// TwinCAT 3 PLC project Untitled1
// ProgramVersion: 3.1.4024.0
// libraries:
//   SysProcess, * (System)
//   Tc2_MC2, * (Beckhoff Automation GmbH)
//   Tc2_Standard, * (Beckhoff Automation GmbH)
//   Tc2_System, * (Beckhoff Automation GmbH)
//   Tc3_MC2_AdvancedHoming, * (Beckhoff Automation GmbH)
//   Tc3_Module, * (Beckhoff Automation GmbH)
//   VisuSymbols,3.5.10.0,System
// project tree:
//   DUTs/ ST_OPCUA.TcDUT
//   / GlobalTextList.TcGTLO, PlcTask.TcTTO, Visualization Manager.TcVMO (not stored)
//   GVLs/ GVL.TcGVL, IO.TcGVL
//   POUs/ Axis.TcPOU, MAIN.TcPOU, POU.TcPOU, process.TcPOU
//   VISUs/ Visualization.TcVIS
// real-time tasks:
//   TASK PlcTask: cycle T#10ms, priority 20, ADS port 350
// motion (NC):
//   TASK NC-Task 1 SAF: cycle T#2ms, priority 4, ADS port 501
//   TASK NC-Task 1 SVB: cycle T#10ms, priority 8, ADS port 511
//   AXIS Axis 1 (id 1)
//     OtherSettings: AllowMotionCmdToSlave=true
//     encoder EncType=1
//     drive DrvType=5
//       Analog: TorqueSetpointScale=10, ScaleFactorActTorque=0.1
//       TimeComp: TaskDelayCycles=1
//     controller CtrType=1
//       CtrPara: PriorControlFactor=1
//         Observer: BandWidth=20
//   AXIS linear Axis 3 (id 3)
//     Dynamic: AccelerationMaximum=50, DecelerationMaximum=50, Acceleration=25, Deceleration=25, Jerk=1211.25
//     Velo: RefSearch=200, RefSync=50, SlowManual=13.4583333333333, FastManual=80.75, Fast=269.166666666667, Maximum=269.167
//     PositionAreaControl: Enable=false
//     TargetPosControl: Enable=false
//     OtherSettings: AllowMotionCmdToSlave=true
//     encoder EncType=19
//       EncPara: ScaleFactorNumerator=10, ScaleFactorDenominator=1048576, MaxCount=#xffffffff
//         SoftEndMinControl: Enable=true
//         SoftEndMaxControl: Enable=true, Range=325
//     drive DrvType=16
//       DrvPara: MaxCount=#xffffffff, DriveControlDWord=#x00020100
//         Analog: VeloReferenz=296.083333333333, VeloScale=32, TorqueSetpointScale=10, ScaleFactorActTorque=0.1
//         TimeComp: TaskDelayCycles=1
//     controller CtrType=1
//       CtrPara: PriorControlFactor=1
//         PosDiffControl: Enable=false
//         Observer: BandWidth=20
//   AXIS rotatioin Axis 4 (id 2)
//     General: UnitName=Degree
//     Dynamic: AccelerationMaximum=150, DecelerationMaximum=150, Acceleration=800.128, Deceleration=800.128, Jerk=7113.39
//     Velo: RefSearch=180, RefSync=5, SlowManual=60, FastManual=180, Fast=29178, Maximum=180
//     PositionAreaControl: Enable=false
//     TargetPosControl: Enable=false
//     OtherSettings: AllowMotionCmdToSlave=true, PulseDistancePos=50, PulseDistanceNeg=50
//     encoder EncType=19
//       EncPara: ScaleFactorNumerator=360, ScaleFactorDenominator=1048576, MaxCount=#xffffffff
//     drive DrvType=16
//       DrvPara: MaxCount=#xffffffff, DriveControlDWord=#x00020100
//         Analog: VeloReferenz=360, TorqueSetpointScale=10, ScaleFactorActTorque=0.1
//         TimeComp: TaskDelayCycles=1
//     controller CtrType=1
//       CtrPara: PriorControlFactor=1
//         PosDiffControl: Enable=false
//         Observer: BandWidth=20
// I/O:
//   DEVICE Device 1 (EtherCAT), AmsNetId 5.143.138.190.2.1
//     Term 12 (EK1200) [EK1200-5000 EtherCAT Power supply (2A E-Bus)]
//       Term 5 (EL7201-0010) [EL7201-0010 1Ch. MDP742 Servo motor output stage with OCT (50V, 2.8A RMS)]
//       Term 6 (EL7201-0010) [EL7201-0010 1Ch. MDP742 Servo motor output stage with OCT (50V, 2.8A RMS)]
//       Term 7 (EL1809) [EL1809 16Ch. Dig. Input 24V, 3ms]
//       Term 8 (EL3356) [EL3356 1Ch. Ana. Input Resistor Bridge Terminal, 16bit, High Precision]
//       Term 12 (EL3064) [EL3064 4Ch. Ana. Input 0-10V]
//       Term 13 (EL3356) [EL3356 1Ch. Ana. Input Resistor Bridge Terminal, 16bit, High Precision]
//       Term 14 (EL3356) [EL3356 1Ch. Ana. Input Resistor Bridge Terminal, 16bit, High Precision]
//       Term 15 (EL1008) [EL1008 8Ch. Dig. Input 24V, 3ms]
//       Term 16 (EL2088) [EL2088 8Ch. Dig. Output 24V, 0.5A, switching to negative]
//       Term 22 (EL9010) [EL9010 End Terminal]
//   DEVICE Device 2 (EtherCAT Automation Protocol), AmsNetId 5.143.138.190.3.1
//   DEVICE Device 3 (EtherCAT Automation Protocol), AmsNetId 5.143.138.190.4.1
// variable links:
//   NC-Task 1 SAF/Axes/linear Axis 3 <-> Device 1 (EtherCAT)/Term 12 (EK1200)/Term 5 (EL7201-0010)
//     Drive/Inputs/In/nDataIn1 <-> DRV Following error actual value/Following error actual value
//     Drive/Inputs/In/nDcOutputTime <-> InfoData/DcOutputShift
//     Drive/Inputs/In/nState1 <-> DRV Statusword/Statusword
//     Drive/Inputs/In/nState2 <-> DRV Statusword/Statusword @bit 8
//     Drive/Inputs/In/nState4 @bit 1 <-> WcState/InputToggle
//     Drive/Inputs/In/nState4 <-> WcState/WcState
//     Drive/Outputs/Out/nCtrl1 <-> DRV Controlword/Controlword
//     Drive/Outputs/Out/nCtrl2 <-> DRV Controlword/Controlword @bit 8
//     Drive/Outputs/Out/nDataOut1 <-> DRV Target position/Target position
//     Enc/Inputs/In/nDataIn1 <-> FB Position/Position
//     Enc/Inputs/In/nDcInputTime <-> InfoData/DcInputShift
//     Enc/Inputs/In/nState4 @bit 1 <-> WcState/InputToggle
//     Enc/Inputs/In/nState4 <-> WcState/WcState
//   NC-Task 1 SAF/Axes/rotatioin Axis 4 <-> Device 1 (EtherCAT)/Term 12 (EK1200)/Term 6 (EL7201-0010)
//     Drive/Inputs/In/nDataIn1 <-> DRV Following error actual value/Following error actual value
//     Drive/Inputs/In/nDcOutputTime <-> InfoData/DcOutputShift
//     Drive/Inputs/In/nState1 <-> DRV Statusword/Statusword
//     Drive/Inputs/In/nState2 <-> DRV Statusword/Statusword @bit 8
//     Drive/Inputs/In/nState4 @bit 1 <-> WcState/InputToggle
//     Drive/Inputs/In/nState4 <-> WcState/WcState
//     Drive/Outputs/Out/nCtrl1 <-> DRV Controlword/Controlword
//     Drive/Outputs/Out/nCtrl2 <-> DRV Controlword/Controlword @bit 8
//     Drive/Outputs/Out/nDataOut1 <-> DRV Target position/Target position
//     Enc/Inputs/In/nDataIn1 <-> FB Position/Position
//     Enc/Inputs/In/nDcInputTime <-> InfoData/DcInputShift
//     Enc/Inputs/In/nState4 @bit 1 <-> WcState/InputToggle
//     Enc/Inputs/In/nState4 <-> WcState/WcState
//   Untitled1/Untitled1 Instance <-> Device 1 (EtherCAT)/Term 12 (EK1200)/Term 16 (EL2088)
//     PlcTask Outputs/IO.cilindertopos1 <-> Channel 6/Output
//     PlcTask Outputs/IO.cilindertopos2 <-> Channel 7/Output
//     PlcTask Outputs/IO.enableledstrip <-> Channel 8/Output
//     PlcTask Outputs/IO.enabletool1 <-> Channel 1/Output
//     PlcTask Outputs/IO.enabletool2 <-> Channel 2/Output
//     PlcTask Outputs/IO.errorlamp <-> Channel 5/Output
//     PlcTask Outputs/IO.initresetlamp <-> Channel 3/Output
//     PlcTask Outputs/IO.processlamp <-> Channel 4/Output
//   Untitled1/Untitled1 Instance <-> Device 1 (EtherCAT)/Term 12 (EK1200)/Term 7 (EL1809)
//     PlcTask Inputs/IO.cilinderpos1 <-> Channel 9/Input
//     PlcTask Inputs/IO.cilinderpos2 <-> Channel 10/Input
//     PlcTask Inputs/IO.doorswitch <-> Channel 11/Input
//     PlcTask Inputs/IO.estop1 <-> Channel 4/Input
//     PlcTask Inputs/IO.estop2 <-> Channel 5/Input
//     PlcTask Inputs/IO.powerok <-> Channel 12/Input
//     PlcTask Inputs/IO.reflinear <-> Channel 13/Input
//     PlcTask Inputs/IO.refrotation <-> Channel 6/Input
//     PlcTask Inputs/IO.resetbutton <-> Channel 3/Input
//     PlcTask Inputs/IO.spare1 <-> Channel 7/Input
//     PlcTask Inputs/IO.spare2 <-> Channel 8/Input
//     PlcTask Inputs/IO.startbutton <-> Channel 16/Input
//     PlcTask Inputs/IO.stopbutton <-> Channel 2/Input
//   Untitled1/Untitled1 Instance <-> NC-Task 1 SAF/Axes/linear Axis 3
//     PlcTask Inputs/MAIN.LinearAxis.axis.NcToPlc <-> Outputs/ToPlc
//     PlcTask Outputs/MAIN.LinearAxis.axis.PlcToNc <-> Inputs/FromPlc
//   Untitled1/Untitled1 Instance <-> NC-Task 1 SAF/Axes/rotatioin Axis 4
//     PlcTask Inputs/MAIN.RotationAxis.axis.NcToPlc <-> Outputs/ToPlc
//     PlcTask Outputs/MAIN.RotationAxis.axis.PlcToNc <-> Inputs/FromPlc

CONFIGURATION Untitled1
    RESOURCE PLC ON TwinCAT3
        TASK PlcTask(INTERVAL := T#10ms, PRIORITY := 20);
        PROGRAM MAIN WITH PlcTask : MAIN;
    END_RESOURCE
END_CONFIGURATION

// ---- DUTs/ST_OPCUA.TcDUT
TYPE ST_OPCUA :
STRUCT	
	nMyNumber : INT;
	bEnable : BOOL;
	sMessage : STRING;
END_STRUCT
END_TYPE

// ---- GVLs/GVL.TcGVL
{attribute 'qualified_only'}
VAR_GLOBAL
END_VAR

// ---- GVLs/IO.TcGVL
{attribute 'qualified_only'}
VAR_GLOBAL
	//Raw value of 3 load cells together
	EL3356_valueX AT %I* : DINT;
	EL3356_valueY AT %I* : DINT;
	EL3356_valueZ AT %I* : DINT;
	
	//inputs
	startbutton AT %I* : BOOL;
	stopbutton AT %I* :BOOL;
	resetbutton AT %I* : BOOL;
	estop1 AT %I* : BOOL; 
	estop2 AT %I* : BOOL; 
	refrotation AT %I* :BOOL;
	spare1 AT %I* :BOOL;
	spare2 AT %I* :BOOL;
	cilinderpos1 AT %I* :BOOL;
	cilinderpos2 AT %I* :BOOL;
	doorswitch AT %I* :BOOL;
	powerok AT %I* :BOOL;
	reflinear AT %I* :BOOL;
	
	//ouputs
	enabletool1 AT %Q* : BOOL;
	enabletool2 AT %Q* : BOOL;
	initresetlamp AT %Q* : BOOL;
	processlamp AT %Q* : BOOL;
	errorlamp AT %Q* : BOOL;
	cilindertopos1 AT %Q* :BOOL;
	cilindertopos2 AT %Q* :BOOL;
	enableledstrip AT %Q* :BOOL;
	
	
	



END_VAR

// ---- POUs/MAIN.TcPOU
PROGRAM MAIN
VAR
	LinearAxis : axis;
	RotationAxis : axis;
	
	linearPos :real;
	linearVel :INT ;
	executeLinearMove :BOOL;
	executehometostop: BOOL;
	linearhomingdone: BOOL;
	linearmovingdone: BOOL;
	linearsearchinghoming: LREAL;
	linearposafterhoming: LREAL;
	
	rotationPos : REAL;
	rotationVel :INT;
	executeRotationMove : BOOL;	
	executehometozero:BOOL;
	rotationhomingdone : BOOL;
	rotationmovingdone: BOOL;
	rotationsearchinghoming: LREAL;
	rotationposafterhoming: lreal;
	
	
	
	enableaxis: BOOL;
	resetaxis : BOOL;
	
	state: INT :=0;

	timer1 : ton;
	timer2 : ton;
	timerstart1: BOOL;
	timerstart2: BOOL;
	timer2reached: BOOL;
	timer1reached: BOOL;
	timertime1: TIME;
	timertime2: TIME;
	elapsedtime1: TIME;
	elapsedtime2: TIME;
	
	//xCordinates :  ARRAY [0..10000] OF REAL := [200,500,540,300,0];
	//rotationpoints :  ARRAY [0..10000] OF REAL;
	//yCordinates :  ARRAY [0..10000] OF REAL;
	arraynumber : INT := 1;
	
	
	//digi intputs
	resetButton: BOOL;
	startbutton: BOOL;
	stopbutton: BOOL; 
	estop1 : BOOL;
	estop2 : BOOL;
	doorswitch :BOOL;
	powerok: BOOL;
	refsensorrotation: BOOL;
	refsensorlinear: BOOL;

	
	tool2posreached: BOOL;
	tool1posreached: BOOL; 
	
	// digi outputs
	enabletool1: BOOL; // relais
	enabletool2: BOOL; // relais
	initresetlamp : BOOL; // lamp
	enableprocesslamp: BOOL; // lamp	
	errorlamp: BOOL;	// lamp
	tool1pos: BOOL; // valve
	tool2pos: BOOL; // valve
	enableledstrip : BOOL; // light for camera
	
	
	// internal variables
	startsecondround: BOOL;
	programstarted:bool:= false;
	
	// vision communication
	takepicturecommand: BOOL;
	searchingForgear : BOOL; // written by vision system | showed in visu
	gearnotfound : BOOL; // written by vision system | showed in visu
	gearfounded :BOOL; // written by vision system | showed in visu
	sendingdata : BOOL; // written by vision system | showed in visu
	coordinatesreceived: BOOL; // written by vision system


(*
	
	{attribute 'OPC.UA.DA':='1'} // Enables a variable for OPC UA
	{attribute 'OPC.UA.DA.StructuredType':='3'} //Enables StructuredType for a STRUCT or a function block
	stOPCUA : ST_OPCUA;
	
	{attribute 'OPC.UA.DA' := '1'} 
	{attribute 'OPC.UA.DA.Access' := '3'} // 0 = none, 1 = read-only, 2 = write access only, 3 = read and write access (default if no tag is used)
	nCounter : INT :=20;

	{attribute 'OPC.UA.DA' := '1'} 
	{attribute 'OPC.UA.DA.Access' := '3'} // 0 = none, 1 = read-only, 2 = write access only, 3 = read and write access (default if no tag is used)
	teller : INT;
	
	{attribute 'OPC.UA.DA' := '1'} 
	{attribute 'OPC.UA.DA.Access' := '3'}
	bStart : BOOL;
	
	{attribute 'OPC.UA.DA' := '1'} 
	jow : BOOL;
	
	
	{attribute 'OPC.UA.DA' := '1'} 
	{attribute 'OPC.UA.DA.Description' := 'My Test Integer Array'} //Sets a text for the OPC UA attribute "Description".
	aMyNumbers : ARRAY[1..5] OF INT;
	
*)

	X_coords: ARRAY[1..9999] OF REAL;   	// Array to store X coordinates
    Y_coords: ARRAY[1..9999] OF REAL;   	// Array to store Y coordinates
	
	status_message 		: STRING(255);  	// Ontvangt status van Python
	next_move		 	: STRING(255);  	// Ontvangt next move van Python
	StartProcess 		: BOOL := FALSE; 	// Variabele om Python te triggeren
	
	Restart				: BOOL;				// Varaiable om alleen de array te verwijderen wanneer proces klaar is
	PulseTimer : TON;      					// Timer voor puls
	i :INT;
END_VAR

(*
IF bStart THEN
	nCounter := nCounter + 1;
END_IF

*)

(*
PulseTimer(IN := StartProcess, PT := T#500MS);

IF PulseTimer.Q THEN
    StartProcess := FALSE; 					// Reset de puls automatisch
END_IF
*)

IF StartProcess AND NOT Restart THEN
    FOR i := 1 TO 9999 DO
        x_coords[i] := 0.0;   				// Stel X-coördinaten in op 0
        y_coords[i] := 0.0;   				// Stel Y-coördinaten in op 0
    END_FOR
END_IF

IF startprocess THEN
	coordinatesreceived := FALSE;
END_IF

IF NOT resetbutton AND NOT programstarted THEN
	state := 0;
ELSIF powerok AND NOT programstarted THEN
	state:= 10;	
END_IF


IF stopbutton THEN
	state := 300;
END_IF

IF estop1 OR estop2 OR NOT doorswitch THEN
	state := 400;
END_IF

CASE state OF
	
	0:
	errorlamp := FALSE;
	timerstart1:=NOT timer1reached;
	timertime1:= T#500MS;
	IF timer1reached THEN
		initresetlamp := NOT initresetlamp;
	END_IF
	IF resetbutton THEN
		state := 10; 
		errorlamp := FALSE;
	END_IF

	10: //waiting for start up program
	programstarted := true;
	initresetlamp := TRUE;
	timerstart1:=TRUE;
	timertime1:= T#3S;
	IF timer1reached THEN
		timerstart1 := FALSE;
		state:= 20;
	END_IF
	
	20: // start resetting axis
	resetaxis:=TRUE;
	
	timerstart1:=TRUE;
	timertime1:= T#2S;
	IF  tool1posreached or true THEN
		timerstart1 := FALSE;
		state:= 30;
	ELSIF timer1reached  THEN
		errorlamp := TRUE;
	END_IF
	
	30: // stop resetting axis
	resetaxis:= FALSE;
	
	timerstart1:=TRUE;
	timertime1:= T#2S;
	IF timer1reached THEN
		timerstart1 := FALSE;
		state:= 40;
	END_IF
	
	40: // enable axis
	enableaxis := TRUE;

	timerstart1:=TRUE;
	timertime1:= T#2S;
	IF timer1reached THEN
		timerstart1 := FALSE;
		state:= 50;
	END_IF
	
	50: // homing axis
	rotationsearchinghoming := 10;
	linearsearchinghoming := 40;
	rotationposafterhoming:= 0;
	linearposafterhoming := 325;
	executehometostop:= TRUE; // for linear axis
	executehometozero:= TRUE; // rotation axis

	IF linearhomingdone AND rotationhomingdone THEN
		state:= 60;

	END_IF
	
	60: // go to start pos
	linearVel := 250;
	rotationvel := 90;
	linearPos := 325;
	rotationpos := 180;
	

	
	(*
	FOR i := 1 TO 10000 DO
    	xcordinates[i] := 0; 
		rotationpoints[i] := 0;
	END_FOR
	*)
	
	timerstart1:=TRUE;
	timertime1:= T#1S;
	
	IF timer1reached THEN
		executeLinearMove := TRUE;
		executerotationmove:= TRUE;	
		state := 61;
		timerstart1 := FALSE;
	END_IF;

	
	61:
	timerstart1:=TRUE;
	timertime1:= T#2S;
	tool1pos:= TRUE; 
	IF timer1reached AND tool1posreached  THEN 
		tool2pos := FALSE;
	
		enabletool1 := FALSE; // for stopping tools after stop button pressed
		//enabletool2 := FALSE;
		
		enabletool2 := FALSE; // disabling tool 2 after the second round
		enableprocesslamp := FALSE; // show that the process is finished
		timerstart1 := FALSE;
		state := 70;			
	END_IF
	
	
	70: // wait until start pos is reached
	IF linearmovingdone AND rotationmovingdone THEN
		executeLinearMove := FALSE;	
		executerotationmove := FALSE;	
		initresetlamp := FALSE; // show that the initialisation is done
		state:= 80;
	END_IF;
	
	80: // wait on start command
	timerstart1:= NOT timer1reached;
	timertime1:= T#500MS;
	IF timer1reached THEN
		enableprocesslamp := NOT enableprocesslamp;
	END_IF	
	
	IF startbutton THEN
		timerstart1 := FALSE;
		enableprocesslamp := TRUE;
		state := 81;
	END_IF
	
	
	81: // delay send take picture command
	timerstart1:=TRUE;
	timertime1:= T#3S;
	
	IF timer1reached THEN
		timerstart1 := FALSE;
		enableledstrip := TRUE;
		StartProcess := TRUE; //command to python
		
		PulseTimer(IN := StartProcess, PT := T#500MS);

		IF PulseTimer.Q THEN
			StartProcess := FALSE; 					// Reset de puls automatisch
			state := 90;
		END_IF
		
		
	END_IF
	
	90: // wait until confirmation receiving coordinates
	IF coordinatesreceived THEN
		takepicturecommand := FALSE;
		enableledstrip := FALSE;
		timerstart1:=TRUE;
		timertime1:= T#2S;
	ELSIF gearnotfound THEN
		enableledstrip := FALSE;
		state := 80;	
	END_IF	
	
	IF timer1reached THEN
		state := 100;
	END_IF
	
	100: // go to working pos
	linearVel := 250;
	rotationvel := 30;
	linearPos := 10;
	rotationpos := 0;
	
	timerstart1:=TRUE;
	timertime1:= T#10MS;
	
	IF timer1reached THEN
		IF NOT startsecondround THEN
			enabletool1 := TRUE;
		END_IF
		executeLinearMove := TRUE;
		executerotationmove:= TRUE;				
		timerstart1 := FALSE;
		state := 110;
	END_IF
	
	
	110: // wait untill working pos is reached
	IF linearmovingdone AND rotationmovingdone THEN
		executeLinearMove := FALSE;	
		executerotationmove := FALSE;	
		state:= 120;
	END_IF;
	
	
	120: // set coordinate pos
	linearVel := 50;
	rotationvel := 30;
	linearPos := x_coords[arraynumber];
	rotationpos := y_coords[arraynumber];
	timerstart1:=TRUE;
	timertime1:= T#10MS;
	
	
	IF timer1reached THEN
		executeLinearMove := TRUE;
		executerotationmove:= TRUE;
		timerstart1 := FALSE;
		state := 130;
	END_IF
	
	130: //execute coordinate pos
	IF linearmovingdone AND rotationmovingdone THEN
		executeLinearMove := FALSE;	
		executerotationmove := FALSE;	
		state:= 120;
		IF (x_coords[arraynumber]) = 0 AND NOT startsecondround THEN
			state := 140;
		ELSIF  (x_coords[arraynumber]) = 0 AND startsecondround THEN
			startsecondround := FALSE;
			state := 60;
		END_IF
		arraynumber := arraynumber +10;	
	END_IF
	
	140: // move away from tool pos
	linearVel := 250;
	rotationvel := 50;
	linearPos := 200;
	rotationpos := 180;
	
	timerstart1:=TRUE;
	timertime1:= T#10MS;
	
	IF timer1reached THEN
		executeLinearMove := TRUE;
		executerotationmove:= TRUE;
		timerstart1 := FALSE;
		state := 160;
	END_IF

	
	160: // wait until away from tool pos is reached and disable tool 1, enanble tool 2, switch tool
	IF linearmovingdone AND rotationmovingdone THEN
		enabletool1 := FALSE;
		enabletool2 := TRUE;
		
		tool1pos := FALSE;
		tool2pos := TRUE;
		timerstart1:=TRUE;
		timertime1:= T#3S;
		
		executeLinearMove := FALSE;	
		executerotationmove := FALSE;	
	END_IF;
	
	IF tool2posreached THEN
		state := 100;
		arraynumber := 1;
		startsecondround := TRUE;
		errorlamp:= false;
	ELSIF timer1reached THEN
		errorlamp:= TRUE;		
	END_IF
	
	
	300: // stop steps
	executeLinearMove := FALSE;	
	executerotationmove := FALSE;	
	
	timerstart1:=TRUE;
	timertime1:= T#10MS;
	
	IF timer1reached THEN
		timerstart1 := FALSE;
		state := 60;
	END_IF
	
	400: //noodstop
	executeLinearMove := FALSE;	
	executerotationmove := FALSE;	
	enabletool1 := FALSE;
	enabletool2 := FALSE;
	errorlamp := TRUE;
	initresetlamp:= FALSE;
	
	timerstart1:=TRUE;
	timertime1:= T#10MS;
	IF timer1reached THEN
		timerstart1:= FALSE;
		state := 0;
	END_IF
END_CASE


LinearAxis(
	enableAxis := enableaxis, 
	executeMove := executeLinearMove, 
	executeHometozero:=  executehometostop,
	pos := linearPos, 
	vel := linearVel, 
	resetaxis := resetaxis,
	refsensor :=NOT refsensorlinear,
	homingsearchvelocity:= linearsearchinghoming,
	posafterhoming:= linearposafterhoming,
	homingDoneTozero => linearhomingdone,
	posreached => linearmovingdone
);

RotationAxis(
	enableAxis := enableaxis, 
	executeMove := executerotationMove, 
	executeHometozero:= executehometozero,
	pos := rotationPos, 
	vel := rotationvel, 
	resetaxis := resetaxis,
	refsensor := refsensorrotation,
	homingsearchvelocity:= rotationsearchinghoming,
	posafterhoming := rotationposafterhoming,
	homingDoneToZero => rotationhomingdone,
	posreached => rotationmovingdone
);

timer2(in := timerstart2, pt := timertime2, et=> elapsedtime1, q=>timer2reached);
timer1(in := timerstart1, pt := timertime1, et=> elapsedtime2, q=> timer1reached);



//	 _ _______                                             _             
//	| (_______)                                        _  (_)            
//	| |_     _     ____ ___  ____  ____  _____  ____ _| |_ _ ____   ____ 
//	| | |   | |   / ___) _ \|  _ \|  _ \| ___ |/ ___|_   _) |  _ \ / _  |
//	| | |___| |  ( (__| |_| | | | | | | | ____( (___  | |_| | | | ( (_| |
//	|_|\_____/    \____)___/|_| |_|_| |_|_____)\____)  \__)_|_| |_|\___ |
//	                                                              (_____|

//inputs
tool1posreached := io.cilinderpos1;
tool2posreached := io.cilinderpos2;
resetbutton := io.resetbutton;
startbutton := io.startbutton;
stopbutton := NOT io.stopbutton;
estop1 := NOT io.estop1;
estop2 := io.estop2;
doorswitch := io.doorswitch;
powerok := io.powerok;
refsensorrotation := io.refrotation;
refsensorlinear := io.reflinear;

//outputs
io.enabletool1 := enabletool1;
io.enabletool2 := enabletool2;
io.cilindertopos1 := tool1pos;
io.cilindertopos2 := tool2pos;
io.initresetlamp:= initresetlamp;
io.processlamp := enableprocesslamp;
io.errorlamp := errorlamp;
io.enableledstrip := enableledstrip;

END_PROGRAM

// ---- POUs/Axis.TcPOU
FUNCTION_BLOCK Axis
VAR_INPUT
	executeMove:BOOL;
	pos :real;
	vel:INT;
	enableAxis : BOOL;
	resetaxis : BOOL;
	executeHomeToStop: BOOL;
	executeHomeToZero : BOOL;
	homingsearchvelocity : LREAL;
	posafterhoming: LREAL;
	refsensor: BOOL;
END_VAR
VAR_OUTPUT
	posreached: BOOL;
	homingDoneToZero: BOOL;
	homingDoneToStop: bool;
	//movingDone: BOOL;
END_VAR
VAR
	axis: AXIS_REF;
	move_abs: MC_moveabsolute;
	power_axis : MC_power;
	reset_axis: MC_reset;
	home_axis: MC_home;
	home_axistostop: MC_stepblock;
	
	homingsettings: ST_HomingOptions;	
	homingparas: mc_homingparameter;
	

END_VAR

power_axis(axis:=axis);
move_abs(axis:=axis);
reset_axis(axis := axis);
home_axis(axis:= axis);
home_axistostop(axis:= axis, parameter := homingparas);



power_axis.Enable := enableAxis;
reset_axis.execute := resetaxis;
move_abs.Velocity := vel;
move_abs.Position := pos;
move_abs.Execute := executeMove;
posreached := move_abs.Done;

power_axis.Enable_Negative:= TRUE;
power_axis.Enable_Positive:= TRUE;

// homing axis with refsensor
home_axis.HomingMode := mc_defaulthoming;
home_axis.Position := posafterhoming; //pos after homing
home_axis.Options := homingsettings;
home_axis.Execute := executeHomeTozero;
home_axis.bCalibrationCam := refsensor; 
homingDoneToZero:= home_axis.Done;

homingsettings.SearchVelocity :=homingsearchvelocity;
homingsettings.SearchDirection := 1; // positive direction

// home axis to endstop
home_axistostop.Execute := executeHomeToStop;
home_axistostop.Direction:= 3;
home_axistostop.Velocity := 30;
home_axistostop.SetPosition := 0;
home_axistostop.DetectionVelocityLimit := 40;
home_axistostop.DetectionVelocityTime:= T#1S;
home_axistostop.TimeLimit := T#20S;
home_axistostop.TorqueLimit:= 200;
home_axistostop.DistanceLimit:=1000;
home_axistostop.TorqueTolerance := 10;
homingDoneTostop := home_axistostop.Done;

END_FUNCTION_BLOCK

// ---- POUs/POU.TcPOU
PROGRAM POU
VAR
	xCordinates :  ARRAY[0..10000] OF INT;
	yCordinates :  ARRAY[0..10000] OF INT;
	mcPower : MC_Power;
	mcSetPosition: MC_SetPosition;
	mcMoveAboslute: MC_MoveAbsolute;
	mcMoveRelative: MC_MoveRelative;
	mcMoveVelocity: MC_MoveVelocity;
	mcReset:MC_Reset;
	mcHalt:MC_Halt;
	mcStop:MC_Stop;
	
	bEnable : BOOL;
	bExecute_SPOS :BOOL;
	bExecute_MABS :BOOL;
	bExecute_MREL :BOOL;
	bExecute_RES :BOOL;
	bExecute_VEL :BOOL;
	bExecute_HALT :BOOL;
	bExecute_STOP :BOOL;
	
	fVelocity:LREAL;
	fPosition:LREAL;
	fAccel:LREAL;
END_VAR

mcPower.Enable:=true;

END_PROGRAM

// ---- POUs/process.TcPOU
FUNCTION_BLOCK process
VAR_INPUT
END_VAR
VAR_OUTPUT
END_VAR
VAR
END_VAR

END_FUNCTION_BLOCK

// ---- VISUs/Visualization.TcVIS
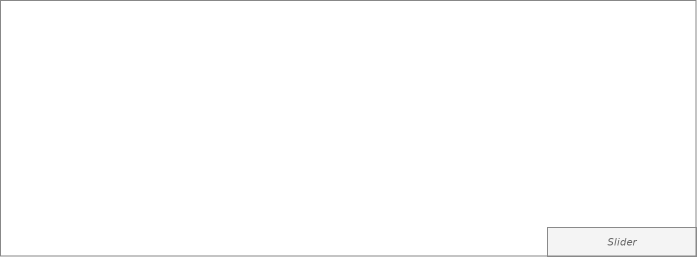
VISUALIZATION Visualization  // 697x257
    Slider (547,227 150x30), variable: MAIN.linearVel, scale 0..20000
END_VISUALIZATION
